METHOD error_reset : BOOL // Must be overrided if future has any errors.
_error_id := _fb_gear_in.ErrorID;
IF _error_id <> 0 THEN
	CASE _reset_state OF
		0:
			_mc_reset(Axis := _axis_main, Execute := FALSE);
			_mc_reset(Axis:= _axis_main, Execute := TRUE );
			_reset_state := 1;
		1:
			IF _mc_reset.Busy THEN
				_mc_reset(Axis:= _axis_main,Execute := FALSE);
			END_IF
			IF _mc_reset.Done AND NOT _mc_reset.Busy THEN
				_reset_state := 2;
			END_IF
		2:
			_mc_reset(Axis := _axis_sub, Execute := FALSE);
			_mc_reset(Axis:= _axis_sub, Execute := TRUE );
			_reset_state := 3;
		3:
			IF _mc_reset.Busy THEN
				_mc_reset(Axis:= _axis_main,Execute := FALSE);
			END_IF
			IF _mc_reset.Done AND NOT _mc_reset.Busy THEN
				_reset_state := 4;
			END_IF
		4:
			_mc_reset(Axis:= _axis_sub,Execute := FALSE);
			error_reset := TRUE;
	END_CASE
ELSE
	error_reset := TRUE;
END_IF
END_METHOD

METHOD execute : BOOL // Return TRUE if finish.
execute := FALSE;
CASE _exec_state OF
	0:
		_fb_gear_in(Master := _axis_main,Slave := _axis_sub,Execute := FALSE);
		_fb_gear_in(
			Execute := TRUE,
			Master := _axis_main,
			Slave := _axis_sub,
			RatioNumerator := _ratio_numerator,
			RatioDenominator := _ratio_denominator,
			Acceleration := _acceleration,
			Deceleration := _deceleration,
			Jerk := _jerk,
			BufferMode := _buffer_mode,
			Options := _option
		);
		_exec_state := 1;
	1:
		IF _fb_gear_in.Busy THEN
			_fb_gear_in(Master := _axis_main,Slave := _axis_sub,Execute := FALSE);
		END_IF
		IF NOT _fb_gear_in.Execute AND NOT _fb_gear_in.Busy THEN
			_exec_state := 2;
		END_IF
	2:
		IF _fb_gear_in.InGear OR _fb_gear_in.Error THEN
			_exec_state := 3;
		END_IF
	3:
		execute := TRUE;
		
END_CASE

IF _error_id = 0 AND _fb_gear_in.ErrorID <> 0 THEN
	_reset_state := 0;
END_IF

_error_id := _fb_gear_in.ErrorID;
END_METHOD

METHOD init : BOOL // Return TRUE if finish.

VAR
	axis: INT;
END_VAR
_exec_state := 0;
_reset_state := 0;
_error_id := _fb_gear_in.ErrorID;
init := TRUE;
END_METHOD

PROPERTY nErrorID : HRESULT
GET
nErrorID := _error_id;
END_GET
SET
END_SET
END_PROPERTY

METHOD set_options : BOOL
VAR_INPUT
	ratio_numerator	: MC_LREAL;
	ratio_denominator	: UINT;
	acceleration	: MC_LREAL;		// Set deceleration in case let moving axis halt.
	deceleration	: MC_LREAL;		// Set deceleration in case let moving axis halt.
	jerk			: MC_LREAL;		// Set jerk in case let moving axis halt.
	buffer_mode : MC_BufferMode;
	option : ST_GearInOptions;
END_VAR
_ratio_numerator	:= ratio_numerator;
_ratio_denominator	:= ratio_denominator;
_acceleration := acceleration;
_deceleration := deceleration;
_jerk := jerk;
_buffer_mode := buffer_mode;
_option := option;
END_METHOD

METHOD set_parameters : BOOL
VAR_INPUT
	axis_main : REFERENCE TO AXIS_REF;
	axis_sub : REFERENCE TO AXIS_REF;

END_VAR
_axis_main REF= axis_main;
_axis_sub REF= axis_sub;
END_METHOD

END_FUNCTION_BLOCK

// ---- POUs/model/activities/FutureMCGearInCreator.TcPOU
FUNCTION_BLOCK FutureMCGearInCreator IMPLEMENTS I_TaskCreator
VAR_INPUT
END_VAR
VAR_OUTPUT
END_VAR
VAR
	_axis_main: REFERENCE TO AXIS_REF;
	_axis_sub: REFERENCE TO AXIS_REF;
	_ratio_numerator	: MC_LREAL := 1;
	_ratio_denominator	: UINT := 1;
	_acceleration: MC_LREAL;
	_deceleration: MC_LREAL;
	_jerk		: MC_LREAL;
	_option : ST_GearInOptions;
	_buffer_mode : MC_BufferMode;
END_VAR

{warning 'add method implementation '}
METHOD create_future : I_Future
VAR_INPUT
	(* Specify future name*)
	future_name	: STRING;
END_VAR
VAR
	_p_future : POINTER TO FutureMCGearIn;
END_VAR
_p_future := __NEW(FutureMCGearIn);
_p_future^.future_name := future_name;
_p_future^.set_parameters(_axis_main, _axis_sub);
_p_future^.set_options(_ratio_numerator, _ratio_denominator, _acceleration, _deceleration,_jerk ,_buffer_mode, _option);
create_future := _p_future^;
END_METHOD

{warning 'add method implementation '}
METHOD destroy_future : I_Future
VAR_INPUT
	(* Specify future instance whtat you want to delete.*)
	future	: I_Future;
END_VAR
VAR
	_p_future : POINTER TO FutureMCGearIn;
END_VAR
IF __QUERYPOINTER(future, _p_future) THEN
	__DELETE(_p_future);
	IF _p_future = 0  THEN
		destroy_future := 0;
	END_IF
END_IF
END_METHOD

METHOD set_options : BOOL
VAR_INPUT
	ratio_numerator	: MC_LREAL;
	ratio_denominator	: UINT;
	acceleration	: MC_LREAL;		// Set deceleration in case let moving axis halt.
	deceleration	: MC_LREAL;		// Set deceleration in case let moving axis halt.
	jerk			: MC_LREAL;		// Set jerk in case let moving axis halt.
	buffer_mode : MC_BufferMode;
	option : ST_GearInOptions;
END_VAR
_ratio_numerator	:= ratio_numerator;
_ratio_denominator	:= ratio_denominator;
_acceleration := acceleration;
_deceleration := deceleration;
_jerk := jerk;
_buffer_mode := buffer_mode;
_option := option;
END_METHOD

METHOD set_parameters : BOOL
VAR_INPUT
	axis_main : REFERENCE TO AXIS_REF;
	axis_sub : REFERENCE TO AXIS_REF;
END_VAR
_axis_main REF= axis_main;
_axis_sub REF= axis_sub;
END_METHOD

END_FUNCTION_BLOCK

// ---- POUs/model/activities/FutureMCGearOut.TcPOU
{attribute 'enable_dynamic_creation'}
FUNCTION_BLOCK FutureMCGearOut EXTENDS FB_AbstructFuture
VAR_INPUT
END_VAR
VAR_OUTPUT
END_VAR
VAR
	_fb_gear_out	: MC_GearOut;
	_mc_reset	: MC_Reset;
	_axis_sub: REFERENCE TO AXIS_REF;
	_ratio_numerator	: MC_LREAL := 1;
	_ratio_denominator	: UINT := 1;
	_option : ST_GearOutOptions;
	_error_id :HRESULT;
	_exec_state : UDINT;
END_VAR

METHOD error_reset : BOOL // Must be overrided if future has any errors.
IF _error_id <> 0 THEN
	CASE _exec_state OF
		0:
			_mc_reset(Axis := _axis_sub, Execute := FALSE);
			_mc_reset(Axis:= _axis_sub, Execute := TRUE );
			_exec_state := 1;
		1:
			IF _mc_reset.Busy THEN
				_mc_reset(Axis:= _axis_sub,Execute := FALSE);
			END_IF
	END_CASE
	
	_error_id := _mc_reset.ErrorID;
	error_reset := _mc_reset.Done;
ELSE
	error_reset := TRUE;
END_IF
END_METHOD

METHOD execute : BOOL // Return TRUE if finish.
execute := FALSE;
CASE _exec_state OF
	0:
		_fb_gear_out(Slave := _axis_sub,Execute := FALSE);
		_fb_gear_out(
			Execute := TRUE,
			Slave := _axis_sub,
			Options := _option
		);
		_exec_state := 1;
	1:
		IF _fb_gear_out.Busy THEN
			_fb_gear_out(Slave := _axis_sub,Execute := FALSE);
		END_IF
		IF NOT _fb_gear_out.Execute AND NOT _fb_gear_out.Busy THEN
			_exec_state := 2;
		END_IF
	2:
		IF _fb_gear_out.Done OR _fb_gear_out.Error THEN
			_exec_state := 3;
		END_IF
	3:
		execute := TRUE;
		
END_CASE

_error_id := _fb_gear_out.ErrorID;
END_METHOD

METHOD init : BOOL // Return TRUE if finish.

VAR
	axis: INT;
END_VAR
_exec_state := 0;
_error_id := _fb_gear_out.ErrorID;
init := TRUE;
END_METHOD

PROPERTY nErrorID : HRESULT
GET
nErrorID := _error_id;
END_GET
SET
END_SET
END_PROPERTY

METHOD set_options : BOOL
VAR_INPUT
	option : ST_GearOutOptions;
END_VAR
_option := option;
END_METHOD

METHOD set_parameters : BOOL
VAR_INPUT
	axis_sub : REFERENCE TO AXIS_REF;
END_VAR
_axis_sub REF= axis_sub;
END_METHOD

END_FUNCTION_BLOCK

// ---- POUs/model/activities/FutureMCGearOutCreator.TcPOU
FUNCTION_BLOCK FutureMCGearOutCreator IMPLEMENTS I_TaskCreator
VAR_INPUT
END_VAR
VAR_OUTPUT
END_VAR
VAR
	_axis_sub: REFERENCE TO AXIS_REF;
	_option : ST_GearOutOptions;
END_VAR

{warning 'add method implementation '}
METHOD create_future : I_Future
VAR_INPUT
	(* Specify future name*)
	future_name	: STRING;
END_VAR
VAR
	_p_future : POINTER TO FutureMCGearOut;
END_VAR
_p_future := __NEW(FutureMCGearOut);
_p_future^.future_name := future_name;
_p_future^.set_parameters(_axis_sub);
_p_future^.set_options(_option);
create_future := _p_future^;
END_METHOD

{warning 'add method implementation '}
METHOD destroy_future : I_Future
VAR_INPUT
	(* Specify future instance whtat you want to delete.*)
	future	: I_Future;
END_VAR
VAR
	_p_future : POINTER TO FutureMCGearOut;
END_VAR
IF __QUERYPOINTER(future, _p_future) THEN
	__DELETE(_p_future);
	IF _p_future = 0  THEN
		destroy_future := 0;
	END_IF
END_IF
END_METHOD

METHOD set_options : BOOL
VAR_INPUT
	option : ST_GearOutOptions;
END_VAR
_option := option;
END_METHOD

METHOD set_parameters : BOOL
VAR_INPUT
	axis_sub : REFERENCE TO AXIS_REF;
END_VAR
_axis_sub REF= axis_sub;
END_METHOD

END_FUNCTION_BLOCK

// ---- POUs/model/activities/FutureMCHalt.TcPOU
{attribute 'enable_dynamic_creation'}
FUNCTION_BLOCK FutureMCHalt EXTENDS FB_AbstructFuture
VAR_INPUT
END_VAR
VAR_OUTPUT
END_VAR
VAR
	_axis: REFERENCE TO AXIS_REF;
	_fb_halt	: MC_Halt;
	_mc_reset	: MC_Reset;
	_deceleration: MC_LREAL;
	_jerk		: MC_LREAL;
	_option : ST_MoveOptions;
	_buffer_mode : MC_BufferMode;
	_error_id :HRESULT;
	_exec_state : UDINT;
END_VAR

METHOD error_reset : BOOL // Must be overrided if future has any errors.
IF _error_id <> 0 THEN
	CASE _exec_state OF
		0:
			_mc_reset(Axis := _axis, Execute := FALSE);
			_mc_reset(Axis:= _axis, Execute := TRUE );
			_exec_state := 1;
		1:
			IF _mc_reset.Busy THEN
				_mc_reset(Axis:= _axis,Execute := FALSE);
			END_IF
	END_CASE
	
	_error_id := _mc_reset.ErrorID;
	error_reset := _mc_reset.Done;
ELSE
	error_reset := TRUE;
END_IF
END_METHOD

METHOD execute : BOOL // Return TRUE if finish.

CASE _exec_state OF
	0:
		_fb_halt(axis := _axis, Execute := FALSE);
		_fb_halt(
			Axis:= _axis,
			Execute := TRUE,
			Jerk := _jerk,
			BufferMode := _buffer_mode,
			Options := _option
		);
		_exec_state := 1;
	1:
		IF _fb_halt.Busy THEN
			_fb_halt(Axis:= _axis,Execute := FALSE);
		END_IF
END_CASE

_error_id := _fb_halt.ErrorID;
execute := _fb_halt.Done OR _fb_halt.Error;
END_METHOD

METHOD init : BOOL // Return TRUE if finish.
_exec_state := 0;
init := TRUE;
END_METHOD

PROPERTY nErrorID : HRESULT
GET
nErrorID := _error_id;
END_GET
SET
END_SET
END_PROPERTY

METHOD set_options : BOOL
VAR_INPUT
	buffer_mode : MC_BufferMode;
	option : ST_MoveOptions;
END_VAR
_buffer_mode := buffer_mode;
_option := option;
END_METHOD

METHOD set_parameters : BOOL
VAR_INPUT
	axis : REFERENCE TO AXIS_REF;
	deceleration	: MC_LREAL;		// Set deceleration in case let moving axis halt.
	jerk			: MC_LREAL;		// Set jerk in case let moving axis halt.
END_VAR
_axis REF= axis;
_deceleration := deceleration;
_jerk := jerk;
END_METHOD

END_FUNCTION_BLOCK

// ---- POUs/model/activities/FutureMCHaltCreator.TcPOU
FUNCTION_BLOCK FutureMCHaltCreator IMPLEMENTS I_TaskCreator
VAR_INPUT
END_VAR
VAR_OUTPUT
END_VAR
VAR
	_axis: REFERENCE TO AXIS_REF;
	_deceleration: MC_LREAL;
	_jerk		: MC_LREAL;
	_option : ST_MoveOptions;
	_buffer_mode : MC_BufferMode;
END_VAR

{warning 'add method implementation '}
METHOD create_future : I_Future
VAR_INPUT
	(* Specify future name*)
	future_name	: STRING;
END_VAR
VAR
	_p_future : POINTER TO FutureMCHalt;
END_VAR
_p_future := __NEW(FutureMCHalt);
_p_future^.future_name := future_name;
_p_future^.set_parameters(_axis, _deceleration, _jerk);
_p_future^.set_options(_buffer_mode, _option);
create_future := _p_future^;
END_METHOD

{warning 'add method implementation '}
METHOD destroy_future : I_Future
VAR_INPUT
	(* Specify future instance whtat you want to delete.*)
	future	: I_Future;
END_VAR
VAR
	_p_future : POINTER TO FutureMCHalt;
END_VAR
IF __QUERYPOINTER(future, _p_future) THEN
	__DELETE(_p_future);
	IF _p_future = 0  THEN
		destroy_future := 0;
	END_IF
END_IF
END_METHOD

METHOD set_options : BOOL
VAR_INPUT
	buffer_mode : MC_BufferMode;
	option : ST_MoveOptions;
END_VAR
_buffer_mode := buffer_mode;
_option := option;
END_METHOD

METHOD set_parameters : BOOL
VAR_INPUT
	axis : REFERENCE TO AXIS_REF;
	deceleration	: MC_LREAL;		// Set deceleration in case let moving axis halt.
	jerk			: MC_LREAL;		// Set jerk in case let moving axis halt.
END_VAR
_axis REF= axis;
_deceleration := deceleration;
_jerk := jerk;
END_METHOD

END_FUNCTION_BLOCK

// ---- POUs/model/activities/FutureMCInching.TcPOU
{attribute 'enable_dynamic_creation'}
FUNCTION_BLOCK FutureMCInching EXTENDS FB_AbstructFuture
VAR_INPUT
END_VAR
VAR_OUTPUT
END_VAR
VAR
	_mc_jog	: MC_Jog;
	_mc_reset	: MC_Reset;
	_abort_executor		: FB_Executor;
	_axis: REFERENCE TO AXIS_REF;
	_direction : BOOL;
	_position : MC_LREAL;
	_velocity : MC_LREAL;
	_acceleration: MC_LREAL;
	_deceleration: MC_LREAL;
	_jerk		: MC_LREAL;
	_mode : E_JogMode ;
	_reset_state : UINT;
	step : UINT;
END_VAR

METHOD error_reset : BOOL // Must be overrided if future has any errors.
VAR_INST
	watch_delay  : TON;
END_VAR
_error_id := _mc_jog.ErrorID;
IF _error_id <> 0 THEN
	CASE _reset_state OF
		0:
			_mc_reset(Axis := _axis, Execute := FALSE);
			_mc_reset(Axis:= _axis, Execute := TRUE );
			watch_delay(IN := FALSE);
			_reset_state := 1;
		1:
			IF _mc_reset.Busy THEN
				_mc_reset(Axis:= _axis,Execute := FALSE);
				_reset_state := 2;
			END_IF
		2:
			IF _error_id = 0 THEN
				error_reset := TRUE;
				_reset_state := 0;
			ELSE
				watch_delay(IN := TRUE, PT := T#1S);
				IF watch_delay.Q THEN
					error_reset := TRUE;
					_reset_state := 0;
				END_IF
			END_IF
	END_CASE
	
	IF _error_id = 0 THEN
		_reset_state := 0;
	END_IF
ELSE
	error_reset := TRUE;
END_IF
END_METHOD

METHOD execute : BOOL // Return TRUE if finish.
CASE step OF
	0:
		_mc_jog(
			JogForward := _direction,
			JogBackwards := NOT _direction,
			Axis := _axis,
			Position := _position,
			Velocity := _velocity,
			Acceleration := _acceleration,
			Deceleration := _deceleration,
			Jerk := _jerk,
			Mode := E_JogMode.MC_JOGMODE_INCHING
		);
		IF _mc_jog.Done OR _mc_jog.Error THEN
			step := 1;
		END_IF

	1:
		_mc_jog(JogForward := FALSE, JogBackwards := FALSE, Axis := _axis);
		execute := TRUE;
		_error_id := _mc_jog.ErrorID;		
END_CASE
END_METHOD

METHOD init : BOOL // Return TRUE if finish.

VAR
	axis: INT;
END_VAR
_reset_state := 0;
_error_id := _mc_jog.ErrorID;
step := 0;
init := TRUE;
END_METHOD

PROPERTY nErrorID : HRESULT
GET
nErrorID := _error_id;
END_GET
SET
END_SET
END_PROPERTY

METHOD set_options : BOOL
VAR_INPUT
	acceleration	: MC_LREAL;		// Set deceleration in case let moving axis halt.
	deceleration	: MC_LREAL;		// Set deceleration in case let moving axis halt.
	jerk			: MC_LREAL;		// Set jerk in case let moving axis halt.
END_VAR
_acceleration := acceleration;
_deceleration := deceleration;
_jerk := jerk;
END_METHOD

METHOD set_parameters : BOOL
VAR_INPUT
	axis : REFERENCE TO AXIS_REF;
	direction : BOOL;
	position : MC_LREAL;
	velocity : MC_LREAL;
END_VAR
_axis REF= axis;
_direction := direction;
_position := position;
_velocity := velocity;
END_METHOD

END_FUNCTION_BLOCK

// ---- POUs/model/activities/FutureMCInchingCreator.TcPOU
FUNCTION_BLOCK FutureMCInchingCreator IMPLEMENTS I_TaskCreator
VAR_INPUT
END_VAR
VAR_OUTPUT
END_VAR
VAR
	_axis: REFERENCE TO AXIS_REF;
	_direction : BOOL;
	_position : MC_LREAL;
	_velocity : MC_LREAL;
	_acceleration: MC_LREAL;
	_deceleration: MC_LREAL;
	_jerk		: MC_LREAL;
END_VAR

{warning 'add method implementation '}
METHOD create_future : I_Future
VAR_INPUT
	(* Specify future name*)
	future_name	: STRING;
END_VAR
VAR
	_p_future : POINTER TO FutureMCInching;
END_VAR
_p_future := __NEW(FutureMCInching);
_p_future^.future_name := future_name;
_p_future^.set_parameters(_axis, _direction, _position, _velocity);
_p_future^.set_options(_acceleration, _deceleration,_jerk );
create_future := _p_future^;
END_METHOD

{warning 'add method implementation '}
METHOD destroy_future : I_Future
VAR_INPUT
	(* Specify future instance whtat you want to delete.*)
	future	: I_Future;
END_VAR
VAR
	_p_future : POINTER TO FutureMCInching;
END_VAR
IF __QUERYPOINTER(future, _p_future) THEN
	__DELETE(_p_future);
	IF _p_future = 0  THEN
		destroy_future := 0;
	END_IF
END_IF
END_METHOD

METHOD set_options : BOOL
VAR_INPUT
	acceleration	: MC_LREAL;		// Set deceleration in case let moving axis halt.
	deceleration	: MC_LREAL;		// Set deceleration in case let moving axis halt.
	jerk			: MC_LREAL;		// Set jerk in case let moving axis halt.
END_VAR
_acceleration := acceleration;
_deceleration := deceleration;
_jerk := jerk;
END_METHOD

METHOD set_parameters : BOOL
VAR_INPUT
	axis : REFERENCE TO AXIS_REF;
	direction : BOOL;
	position : MC_LREAL;
	velocity : MC_LREAL;
END_VAR
_axis REF= axis;
_direction := direction;
_position := position;
_velocity := velocity;
END_METHOD

END_FUNCTION_BLOCK

// ---- POUs/model/activities/FutureMCPowerCreator.TcPOU
FUNCTION_BLOCK FutureMCPowerCreator IMPLEMENTS I_TaskCreator
VAR_INPUT
END_VAR
VAR_OUTPUT
END_VAR
VAR
	_axis: REFERENCE TO AXIS_REF;
	_override: LREAL := 100.0;
	_enable_positive:	BOOL := TRUE; 
	_enable_negative:	BOOL := TRUE;
	_option : ST_PowerOptions;
	_buffer_mode : MC_BufferMode;
	_status : BOOL;
END_VAR

METHOD create_future : I_Future
VAR_INPUT
	(* Specify future name*)
	future_name	: STRING;
END_VAR
VAR
	_p_future : POINTER TO FutureMCPower;
END_VAR
_p_future := __NEW(FutureMCPower);
_p_future^.future_name := future_name;
_p_future^.set_parameters(_axis, _status);
_p_future^.set_options(_enable_positive, _enable_negative, _override, _buffer_mode, _option);
create_future := _p_future^;
END_METHOD

METHOD destroy_future : I_Future
VAR_INPUT
	(* Specify future instance whtat you want to delete.*)
	future	: I_Future;
END_VAR
VAR
	_p_future : POINTER TO FutureMCPower;
END_VAR
IF __QUERYPOINTER(future, _p_future) THEN
	__DELETE(_p_future);
	IF _p_future = 0  THEN
		destroy_future := 0;
	END_IF
END_IF
END_METHOD

METHOD set_options : BOOL
VAR_INPUT
	Enable_Positive:	BOOL; 
	Enable_Negative:	BOOL;
	Override:			LREAL := 100;
	buffer_mode : MC_BufferMode;
	option : ST_PowerOptions;
END_VAR
_override := Override;
_enable_positive := Enable_Positive;
_enable_negative := Enable_Negative;
_buffer_mode := buffer_mode;
_option := option;
END_METHOD

METHOD set_parameters : BOOL
VAR_INPUT
	axis : REFERENCE TO AXIS_REF;
	status : BOOL;
END_VAR
_axis REF= axis;
_status := status;
END_METHOD

END_FUNCTION_BLOCK

// ---- POUs/model/activities/FutureMCReset.TcPOU
{attribute 'enable_dynamic_creation'}
FUNCTION_BLOCK FutureMCReset EXTENDS FB_AbstructFuture
VAR_INPUT
END_VAR
VAR_OUTPUT
END_VAR
VAR
	_axis: REFERENCE TO AXIS_REF;
	_mc_reset	: MC_Reset;
	_error_id :HRESULT;
	_exec_state : UDINT;
END_VAR

METHOD execute : BOOL // Return TRUE if finish.

CASE _exec_state OF
	0:
		_mc_reset(axis := _axis, Execute := FALSE);
		_mc_reset(Axis:= _axis, Execute := TRUE );
		_exec_state := 1;
	1:
		IF _mc_reset.Busy THEN
			_mc_reset(Axis:= _axis,Execute := FALSE);
		END_IF
END_CASE

_error_id := _mc_reset.ErrorID;
execute := _mc_reset.Done OR _mc_reset.Error;
END_METHOD

METHOD init : BOOL // Return TRUE if finish.
_exec_state := 0;
init := TRUE;
END_METHOD

PROPERTY nErrorID : HRESULT
GET
nErrorID := _error_id;
END_GET
SET
END_SET
END_PROPERTY

METHOD set_parameters : BOOL
VAR_INPUT
	axis : REFERENCE TO AXIS_REF;
END_VAR
_axis REF= axis;
END_METHOD

END_FUNCTION_BLOCK

// ---- POUs/model/activities/FutureMCResetCreator.TcPOU
FUNCTION_BLOCK FutureMCResetCreator IMPLEMENTS I_TaskCreator
VAR_INPUT
END_VAR
VAR_OUTPUT
END_VAR
VAR
	_axis: REFERENCE TO AXIS_REF;
END_VAR

{warning 'add method implementation '}
METHOD create_future : I_Future
VAR_INPUT
	(* Specify future name*)
	future_name	: STRING;
END_VAR
VAR
	_p_future : POINTER TO FutureMCReset;
END_VAR
_p_future := __NEW(FutureMCReset);
_p_future^.future_name := future_name;
_p_future^.set_parameters(_axis);
create_future := _p_future^;
END_METHOD

{warning 'add method implementation '}
METHOD destroy_future : I_Future
VAR_INPUT
	(* Specify future instance whtat you want to delete.*)
	future	: I_Future;
END_VAR
VAR
	_p_future : POINTER TO FutureMCReset;
END_VAR
IF __QUERYPOINTER(future, _p_future) THEN
	__DELETE(_p_future);
	IF _p_future = 0  THEN
		destroy_future := 0;
	END_IF
END_IF
END_METHOD

METHOD set_parameters : BOOL
VAR_INPUT
	axis : REFERENCE TO AXIS_REF;
END_VAR
_axis REF= axis;
END_METHOD

END_FUNCTION_BLOCK

// ---- POUs/model/activities/FutureMCSetPosition.TcPOU
{attribute 'enable_dynamic_creation'}
FUNCTION_BLOCK FutureMCSetPosition EXTENDS FB_AbstructFuture
VAR_INPUT
END_VAR
VAR_OUTPUT
END_VAR
VAR
	_fb_set_position	: MC_SetPosition;
	_mc_reset	: MC_Reset;
	_axis: REFERENCE TO AXIS_REF;
	_position	: MC_LREAL;
	_mode		: BOOL;
	_option 	: ST_SetPositionOptions;
	_error_id :HRESULT;
	_exec_state : UDINT;
	_reset_state : UDINT;
END_VAR

METHOD error_reset : BOOL // Must be overrided if future has any errors.
VAR_INST
	watch_delay  : TON;
END_VAR
_error_id := _fb_set_position.ErrorID;
IF _error_id <> 0 THEN
	CASE _reset_state OF
		0:
			_mc_reset(Axis := _axis, Execute := FALSE);
			_mc_reset(Axis:= _axis, Execute := TRUE );
			watch_delay(IN := FALSE);
			_reset_state := 1;
		1:
			IF _mc_reset.Done THEN
				_mc_reset(Axis:= _axis,Execute := FALSE);
				_reset_state := 2;
			END_IF
		2:
			error_reset := TRUE;
			watch_delay(IN := TRUE, PT := T#1S);
			IF watch_delay.Q THEN
				_reset_state := 0;
			END_IF
	END_CASE
	
	IF _error_id = 0 THEN
		_reset_state := 0;
	END_IF
ELSE
	error_reset := TRUE;
END_IF
END_METHOD

METHOD execute : BOOL // Return TRUE if finish.

CASE _exec_state OF
	0:
		_fb_set_position( Axis:= _axis, Execute := FALSE);
		_fb_set_position(
				Axis := _axis,
				Execute := TRUE, 
				Position := _position,
				Mode := _mode,
				Options := _option
		);
		_exec_state := 1;
	1:
		IF _fb_set_position.Busy THEN
			_fb_set_position( Axis:= _axis, Execute := FALSE);
		END_IF
END_CASE

_error_id := _fb_set_position.ErrorID;
execute := _fb_set_position.Done OR _fb_set_position.Error;
END_METHOD

METHOD init : BOOL // Return TRUE if finish.
_exec_state := 0;
init := TRUE;
END_METHOD

PROPERTY nErrorID : HRESULT
GET
nErrorID := _error_id;
END_GET
SET
END_SET
END_PROPERTY

METHOD set_options : BOOL
VAR_INPUT
	mode		: BOOL;
	option 	: ST_SetPositionOptions;
END_VAR
_mode := mode;
_option := option;
END_METHOD

METHOD set_parameters : BOOL
VAR_INPUT
	axis: REFERENCE TO AXIS_REF;
	position	: MC_LREAL;
END_VAR
_axis REF= axis;
_position := position;
END_METHOD

END_FUNCTION_BLOCK

// ---- POUs/model/activities/FutureMCSetPositionCreator.TcPOU
FUNCTION_BLOCK FutureMCSetPositionCreator IMPLEMENTS I_TaskCreator
VAR_INPUT
END_VAR
VAR_OUTPUT
END_VAR
VAR
	_axis: REFERENCE TO AXIS_REF;
	_position	: MC_LREAL;
	_mode		: BOOL;
	_option 	: ST_SetPositionOptions;
	_error_id :UDINT;
END_VAR

{warning 'add method implementation '}
METHOD create_future : I_Future
VAR_INPUT
	(* Specify future name*)
	future_name	: STRING;
END_VAR
VAR
	_p_future : POINTER TO FutureMCSetPosition;
END_VAR
_p_future := __NEW(FutureMCSetPosition);
_p_future^.future_name := future_name;
_p_future^.set_parameters(_axis, _position);
_p_future^.set_options(_mode, _option);
create_future := _p_future^;
END_METHOD

{warning 'add method implementation '}
METHOD destroy_future : I_Future
VAR_INPUT
	(* Specify future instance whtat you want to delete.*)
	future	: I_Future;
END_VAR
VAR
	_p_future : POINTER TO FutureMCSetPosition;
END_VAR
IF __QUERYPOINTER(future, _p_future) THEN
	__DELETE(_p_future);
	IF _p_future = 0  THEN
		destroy_future := 0;
	END_IF
END_IF
END_METHOD

METHOD set_options : BOOL
VAR_INPUT
	mode		: BOOL;
	option 	: ST_SetPositionOptions;
END_VAR
_mode := mode;
_option := option;
END_METHOD

METHOD set_parameters : BOOL
VAR_INPUT
	axis: REFERENCE TO AXIS_REF;
	position	: MC_LREAL;
END_VAR
_axis REF= axis;
_position := position;
END_METHOD

END_FUNCTION_BLOCK

// ---- POUs/model/activities/FutureTimerBlink.TcPOU
{attribute 'enable_dynamic_creation'}
FUNCTION_BLOCK FutureTimerBlink EXTENDS FB_AbstructFuture
VAR_INPUT
END_VAR
VAR_OUTPUT
END_VAR
VAR
	process_timer: TON;
	blink_timer: TON;
	_set_time :TIME;
	_result :UDINT;
	_output: REFERENCE TO BOOL;
	_process_time: TIME;
	_error_test :BOOL;
END_VAR

METHOD abort : BOOL
IF process_timer.IN THEN
	_set_time := process_timer.PT - process_timer.ET;
END_IF
process_timer(IN := FALSE);
_output := FALSE;
abort := TRUE;
END_METHOD

METHOD error_reset : BOOL // Must be overrided if future has any errors.
_error_test := FALSE;
_result := 0;
error_reset := TRUE;
END_METHOD

PROPERTY error_test : BOOL
SET
_error_test := error_test;
END_SET
END_PROPERTY

METHOD execute : BOOL
VAR_INPUT
END_VAR
blink_timer(IN := NOT blink_timer.Q, PT := T#0.5S);
IF _output AND blink_timer.Q THEN
	_output := FALSE;
ELSIF blink_timer.Q THEN
	_output := TRUE;
END_IF
process_timer(IN := TRUE,PT := _process_time);
execute := process_timer.Q;

IF _error_test THEN
	_result := 9;
	execute := TRUE;
END_IF
END_METHOD

METHOD init : BOOL
VAR_INPUT
END_VAR
_output := FALSE;
_set_time := _process_time;
process_timer(IN := FALSE);
blink_timer(IN := FALSE);
init := TRUE;
END_METHOD

PROPERTY nErrorID : HRESULT
GET
END_GET
END_PROPERTY

METHOD quit : BOOL
THIS^.init();
quit := TRUE;
END_METHOD

METHOD set_options : BOOL
VAR_INPUT
	error_test: BOOL;
END_VAR
_error_test := error_test;
END_METHOD

METHOD set_parameter : BOOL
VAR_INPUT
	process_time: TIME;
	output		: REFERENCE TO BOOL;
END_VAR
_process_time := process_time;
_output REF= output;
END_METHOD

END_FUNCTION_BLOCK

// ---- POUs/model/activities/FutureTimerBlinkCreator.TcPOU
FUNCTION_BLOCK FutureTimerBlinkCreator IMPLEMENTS I_TaskCreator
VAR_INPUT
END_VAR
VAR_OUTPUT
END_VAR
VAR
	_output: REFERENCE TO BOOL;
	_process_time: TIME;
	_error_test :BOOL;
END_VAR

{warning 'add method implementation '}
METHOD create_future : I_Future
VAR_INPUT
	future_name	: STRING;
END_VAR
VAR
	_p_future : POINTER TO FutureTimerBlink;
END_VAR
_p_future := __NEW(FutureTimerBlink);
_p_future^.future_name := future_name;
_p_future^.set_parameter(_process_time, _output);
_p_future^.set_options(_error_test);
create_future := _p_future^;
END_METHOD

{warning 'add method implementation '}
METHOD destroy_future : I_Future
VAR_INPUT
	future	: I_Future;
END_VAR
VAR
	_p_future : POINTER TO FutureTimerBlink;
END_VAR
IF __QUERYPOINTER(future, _p_future) THEN
	__DELETE(_p_future);
	IF _p_future = 0  THEN
		destroy_future := 0;
	END_IF
END_IF
END_METHOD

METHOD set_options : BOOL
VAR_INPUT
	error_test: BOOL;
END_VAR
_error_test := error_test;
END_METHOD

METHOD set_parameter : BOOL
VAR_INPUT
	process_time: TIME;
	output		: REFERENCE TO BOOL;
END_VAR
_process_time := process_time;
_output REF= output;
END_METHOD

END_FUNCTION_BLOCK

// ---- POUs/test/FB_TaskRunner_Test.TcPOU
FUNCTION_BLOCK FB_TaskRunner_Test EXTENDS TcUnit.FB_TestSuite
VAR_INPUT
END_VAR
VAR_OUTPUT
END_VAR
VAR
	runner : FB_TaskRunner;
	fbJobTreeSearch : FB_ExecutorTreeSearch;

	init: BOOL;
	_state :UINT;
	mc_power : FutureMCPower;
	_poweron_job	: FB_Executor;
	
	demo_job	: FB_Executor;
	axis1	: AXIS_REF;
	bPower : BOOL;
	bStart : BOOL;
	
	await : BOOL;
	
	fbGetTimeZoneInformation	: FB_GetTimeZoneInformation := (bExecute := TRUE);
	localTime : FB_LocalSystemTime := (bEnable := TRUE);
	tzinfo : FB_GetTimeZoneInformation := (bExecute := TRUE);
	getSystemtime : FB_TzSpecificLocalTimeToSystemTime;
	current_time : T_FILETIME64;
	observer : REFERENCE TO FB_JobEventLogStr;
	
	motion_data : ST_MotionData;
END_VAR

_01_WhenTaskSpawned();

METHOD PRIVATE _01_WhenTaskSpawned
VAR_INST
	SpecificNumOfJobs : UDINT := 32;
	num_of_jobs : UDINT;
END_VAR

VAR
	state_expect: E_FUTUREEXECUTIONSTATE;
	state_actual: E_FutureExecutionState;
END_VAR
TEST('_01_WhenTaskSpawned');

IF NOT init THEN
	JobCreateDemo(demo_job, axis1); // demo_job にメソッドを通してシーケンスジョブを組み立てる
	mc_power.future_name := 'POWER_CTRL';
	_poweron_job.future := mc_power;
	observer REF= runner.job_event_log_str;
	num_of_jobs := demo_job.children.num_of_jobs;
	init := TRUE;	// RUN 後 1 サイクルだけ実行
END_IF

AssertEquals(
	Expected := SpecificNumOfJobs, 
	Actual := num_of_jobs, 
	Message := 'Test $'Task Spawned$' failed at $'Num of jobs$''
);

state_expect := E_FutureExecutionState.init;
state_actual := demo_job.current_state;



AssertEquals(
	Expected := state_expect, 
	Actual := state_actual, 
	Message := 'Test $'Task Spawned$' failed at $'Num of jobs$''
);

TEST_FINISHED();
END_METHOD

METHOD JobCreateDemo : BOOL
VAR_INPUT
	base_job : REFERENCE TO FB_Executor;
	stAxis1	: REFERENCE TO AXIS_REF;
END_VAR
VAR
	_job_temp : REFERENCE TO FB_Executor;
	_job_temp_parent : REFERENCE TO FB_Executor;
	sleep : POINTER TO FutureSleep;
	sleep_creator : FutureSleepCreator;

	mc_move_rel_future : POINTER TO FutureMCMoveRelative;
	mc_move_rel_future_creator : FutureMCMoveRelativeCreator;

	mc_move_abs_future : POINTER TO FutureMCMoveAbsolute;
	mc_move_abs_future_creator : FutureMCMoveAbsoluteCreator;

	mc_move_velocity_future: POINTER TO FutureMCMoveVelocity;
	mc_move_velocity_future_creator: FutureMCMoveVelocityCreator;
	
	mc_stop_future_creator : FutureMcStopCreator;
	
	i : UDINT;

END_VAR
base_job.create_container(ContainerTYpe.BATCH, 'DEMO_JOB');
// Sequence
_job_temp_parent REF= base_job.children.create_container(ContainerTYpe.BATCH, 'STEP MOVING');
FOR i := 1 TO 10 DO

	mc_move_rel_future_creator.set_parameters(stAxis1,20,200,0,0,0,0);
	_job_temp REF= _job_temp_parent.children.create_job(mc_move_rel_future_creator,'Move +20 deg, 200 deg/s');

	sleep_creator.sleep_time := T#100MS;
	_job_temp REF= _job_temp_parent.children.create_job(sleep_creator,'Wait 100ms');
	
END_FOR

// position set to 0

mc_move_abs_future_creator.set_parameters(stAxis1,0,200,0,0,0,0);
_job_temp REF= base_job.children.create_job(mc_move_abs_future_creator,'Back to home');

FOR i := 1 TO 10 DO

	mc_move_rel_future_creator.set_parameters(stAxis1,-20,200,0,0,0,0);
	_job_temp REF= base_job.children.create_job(mc_move_rel_future_creator,'Move -20 deg, 200 deg/s');

	sleep_creator.sleep_time := T#100MS;
	_job_temp REF= base_job.children.create_job(sleep_creator,'Wait 100ms');
	
END_FOR

// position to 0

mc_move_abs_future_creator.set_parameters(stAxis1,0,200,0,0,0,0);
_job_temp REF= base_job.children.create_job(mc_move_abs_future_creator,'Back to home');

sleep_creator.sleep_time := T#100MS;
_job_temp REF= base_job.children.create_job(sleep_creator,'Wait 100ms');

// 1000deg/s -> 500deg/s

mc_move_velocity_future_creator.set_parameters(stAxis1,MC_Direction.MC_Positive_Direction,1000,0,0,0,0);
_job_temp REF= base_job.children.create_job(mc_move_velocity_future_creator,'Move velocity');

sleep_creator.sleep_time := T#5S;
_job_temp REF= base_job.children.create_job(sleep_creator,'1000 deg/s 5 seconds');

mc_move_velocity_future_creator.set_parameters(stAxis1,MC_Direction.MC_Positive_Direction,500,0,0,0,0);
_job_temp REF= base_job.children.create_job(mc_move_velocity_future_creator,'Move velocity');

sleep_creator.sleep_time := T#5S;
_job_temp REF= base_job.children.create_job(sleep_creator,'500 deg/s 5 seconds');

mc_move_velocity_future_creator.set_parameters(stAxis1,MC_Direction.MC_Positive_Direction,250,0,0,0,0);
_job_temp REF= base_job.children.create_job(mc_move_velocity_future_creator,'Move velocity');

sleep_creator.sleep_time := T#5S;
_job_temp REF= base_job.children.create_job(sleep_creator,'250 deg/s 5 seconds');


mc_stop_future_creator.set_parameters(stAxis1,0,0);
_job_temp REF= base_job.children.create_job(mc_stop_future_creator,'STOP');

// position to 0

mc_move_abs_future_creator.set_parameters(stAxis1,0,1000,0,0,0,0);
_job_temp REF= base_job.children.create_job(mc_move_abs_future_creator,'Back to home');
END_METHOD

END_FUNCTION_BLOCK

// ---- POUs/test/UnitTest.TcPOU
PROGRAM UnitTest
VAR
	fbTaskRunner_Test : FB_TaskRunner_Test;
END_VAR

TcUnit.RUN();

END_PROGRAM

// ---- GlobalTextList.TcGTLO
TEXTLIST GlobalTextList
  467 = '%'
  447 = '%.2f'
  487 = '%0d'
  815 = '%1d'
  505 = '%d'
  805 = '%s'
  276 = 'Job'
  57 = 'Job clear'
  255 = 'Label'
  430 = 'Pause'
  54 = 'Position'
  844 = 'Power'
  592 = 'Process'
  165 = 'Resume'
  119 = 'Speed'
  762 = 'Start'
  363 = 'Status'
  539 = 'Step'
END_TEXTLIST

// ---- VISUs/Visualization.TcVIS
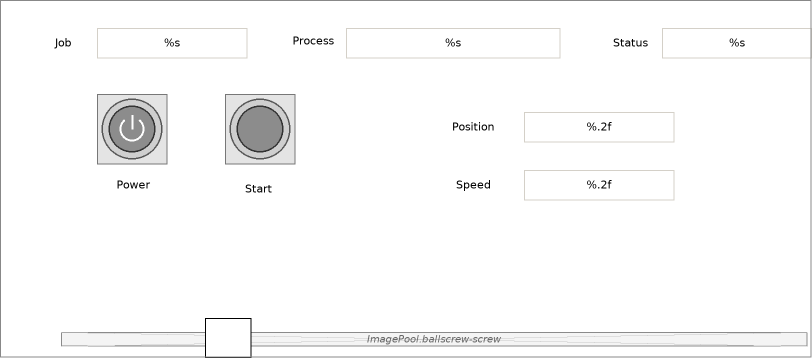
VISUALIZATION Visualization  // 812x358
    PushSwitch (225,94 70x70), variable: demo3.bStart, behaviour: TOGGLE, style: Switch-PushSwitch-Gray
    Textfield (97,28 150x30), "%s", text variable: demo3.runner.job_event_cyclic_output.event_message.job_id
    Label (280,26 67x30), "Process"
    Label (30,28 67x30), "Job"
    PowerSwitch (97,94 70x70), variable: demo3.bPower, behaviour: TOGGLE, style: Switch-PowerSwitch-Gray
    Textfield (524,112 150x30), "%.2f", text variable: GVL.axis1.NcToPlc.ActPos
    Textfield (346,28 214x30), "%s", text variable: demo3.runner.job_event_cyclic_output.event_message.subject
    Textfield (662,28 150x30), "%s", text variable: demo3.runner.job_event_cyclic_output.event_message.new_state
    Label (597,28 67x30), "Status"
    Textfield (524,170 150x30), "%.2f", text variable: GVL.axis1.NcToPlc.ActVelo
    Image (61,332 746x14), image: ImagePool.ballscrew-screw
    Rectangle (205,318 46x40)
        p3560616238: GVL.axis1.NcToPlc.ActPos / 10.0
    Label (100,170 67x30), "Power"
    Label (225,174 67x30), "Start"
    Label (440,112 67x30), "Position"
    Label (440,170 67x30), "Speed"
END_VISUALIZATION
